// TIA Portal V15.1 export
// export: Created 2024-06-21T08:41:25.533852Z, ExportSetting WithDefaults, DisplayName Totally Integrated Automation Portal, DisplayVersion V15.1 Update 5, DisplayName TIA Portal Openness, DisplayVersion V15.1 Update 5, DisplayName SINAMICS Startdrive Advanced, DisplayVersion V15.1, DisplayName G130, G150, S120, S150, SINAMICS MV, S210, DisplayVersion V15.1, DisplayName G110M, G120, G120C, G120D, G120P, DisplayVersion V15.1, DisplayName STEP 7 Professional, DisplayVersion V15.1 Update 5, DisplayName STEP 7 Safety, DisplayVersion V15.1, DisplayName WinCC Professional, DisplayVersion V15.1 Update 5, DisplayName SIMATIC Visualization Architect, DisplayVersion V15.1
FUNCTION "PNComPLC308" : Void   // FC260, FBD
TITLE = PNComPLC308
{ S7_Optimized_Access := 'FALSE' }
AUTHOR : VCG
FAMILY : LocFncGn
NAME : 211Intf
VERSION : 0.1
// stored: AutoNumber false, IsIECCheckEnabled false, SetENOAutomatically False, UDAEnableTagReadback false
   VAR_OUTPUT
      O_AlarmA : Bool;   // Alarm A
      O_AlarmB : Bool;   // Alarm B
      O_AlarmC : Bool;   // Alarm C
      O_AlarmD : Bool;   // Alarm D
      O_AlarmABCondition : Bool;   // Alarms resetable
      H_IAnim : Word;   // For animation of icon
   END_VAR
BEGIN

REGION Network 1: **** --------------------- 308240CR27 --> 210CR21 --------------------- ****
END_REGION

REGION Network 2: **** 1 - Inputs **** 308230ZS01 - Access Stop Request
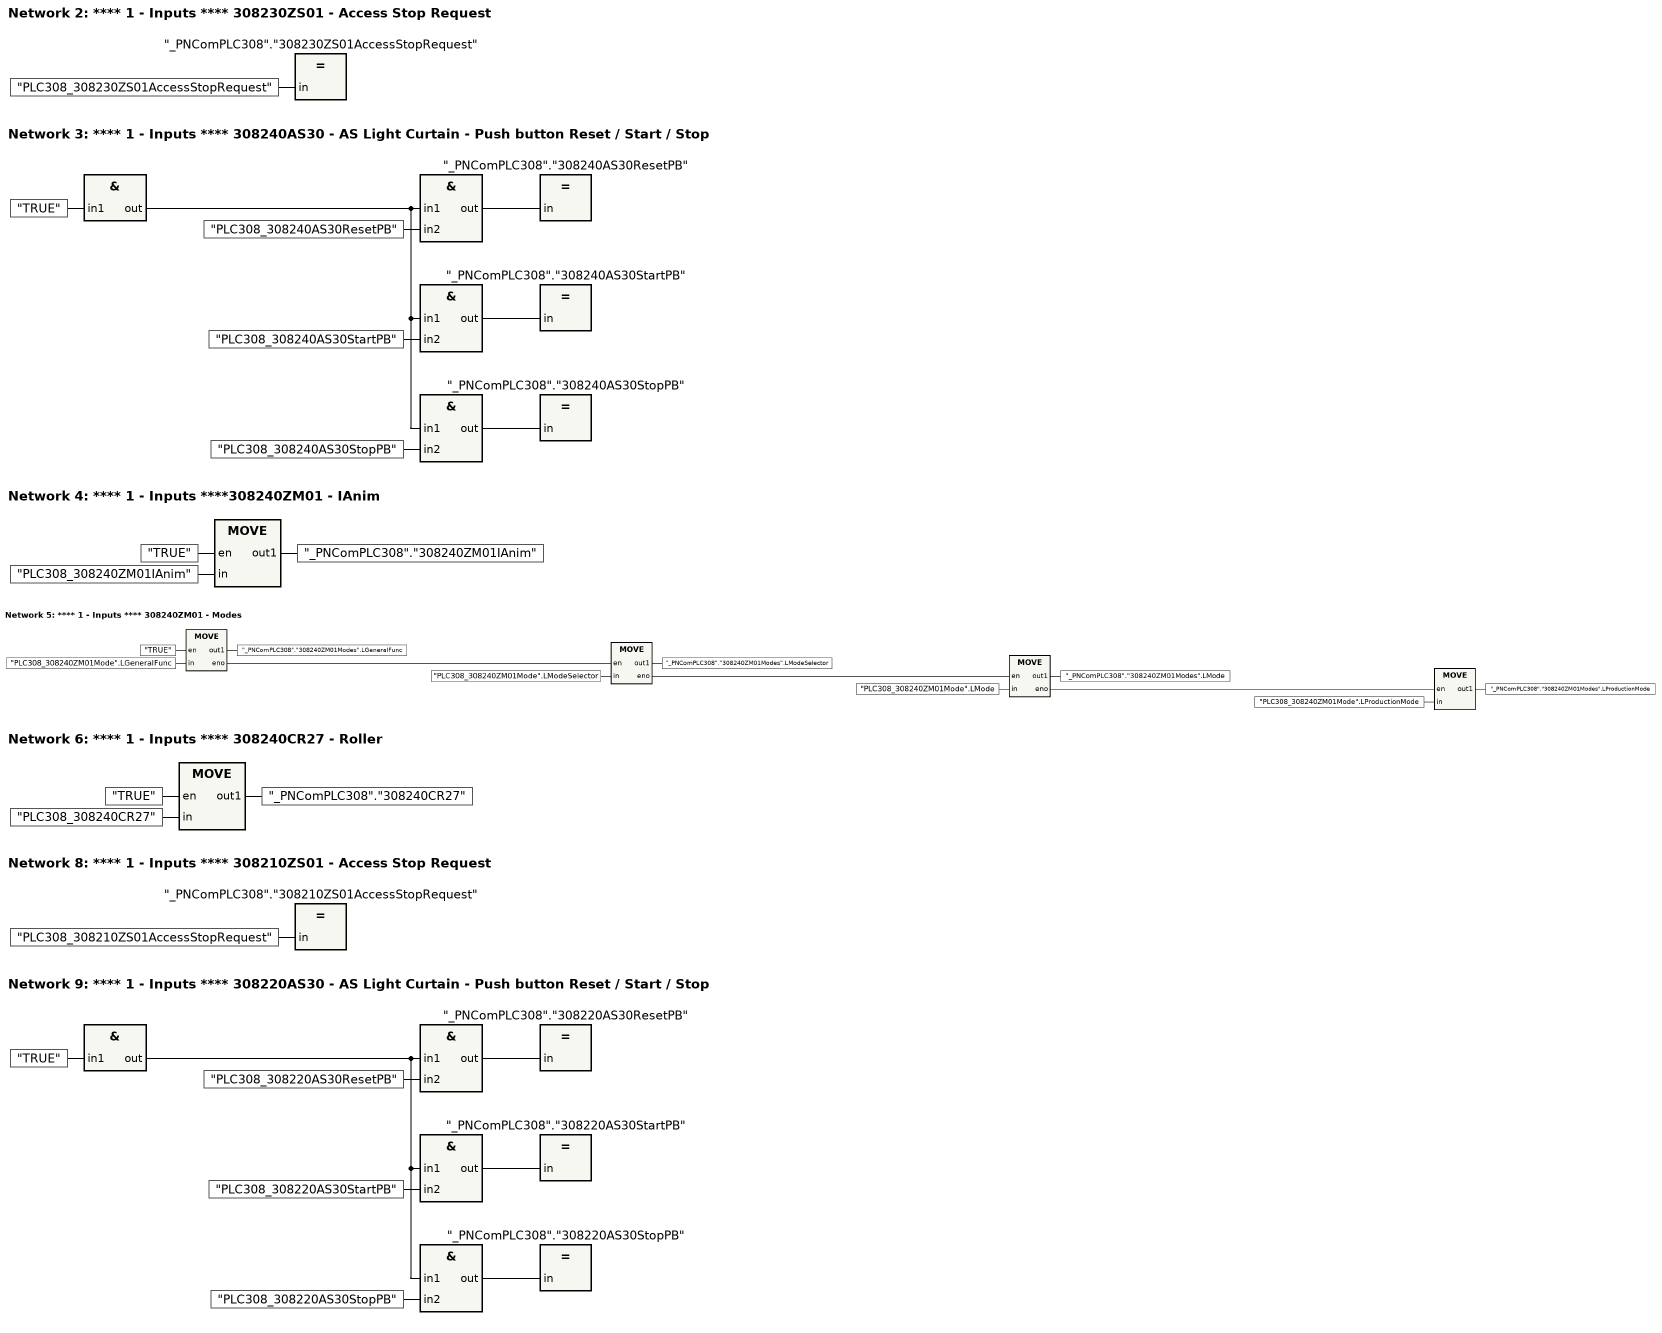
   "_PNComPLC308"."308230ZS01AccessStopRequest" := "PLC308_308230ZS01AccessStopRequest";
END_REGION

REGION Network 3: **** 1 - Inputs **** 308240AS30 - AS Light Curtain - Push button Reset / Start / Stop
   "_PNComPLC308"."308240AS30ResetPB" := "TRUE" AND "PLC308_308240AS30ResetPB";
   "_PNComPLC308"."308240AS30StartPB" := "TRUE" AND "PLC308_308240AS30StartPB";
   "_PNComPLC308"."308240AS30StopPB" := "TRUE" AND "PLC308_308240AS30StopPB";
END_REGION

REGION Network 4: **** 1 - Inputs ****308240ZM01 - IAnim
   IF "TRUE" THEN "_PNComPLC308"."308240ZM01IAnim" := "PLC308_308240ZM01IAnim"; END_IF;
END_REGION

REGION Network 5: **** 1 - Inputs **** 308240ZM01 - Modes
   IF "TRUE" THEN
       "_PNComPLC308"."308240ZM01Modes".LGeneralFunc := "PLC308_308240ZM01Mode".LGeneralFunc;
       "_PNComPLC308"."308240ZM01Modes".LModeSelector := "PLC308_308240ZM01Mode".LModeSelector;
       "_PNComPLC308"."308240ZM01Modes".LMode := "PLC308_308240ZM01Mode".LMode;
       "_PNComPLC308"."308240ZM01Modes".LProductionMode := "PLC308_308240ZM01Mode".LProductionMode;
   END_IF;
END_REGION

REGION Network 6: **** 1 - Inputs **** 308240CR27 - Roller
   IF "TRUE" THEN "_PNComPLC308"."308240CR27" := "PLC308_308240CR27"; END_IF;
END_REGION

REGION Network 7: **** --------------------- 308220CR28 --> 220CR21 --------------------- ****
END_REGION

REGION Network 8: **** 1 - Inputs **** 308210ZS01 - Access Stop Request
   "_PNComPLC308"."308210ZS01AccessStopRequest" := "PLC308_308210ZS01AccessStopRequest";
END_REGION

REGION Network 9: **** 1 - Inputs **** 308220AS30 - AS Light Curtain - Push button Reset / Start / Stop
   "_PNComPLC308"."308220AS30ResetPB" := "TRUE" AND "PLC308_308220AS30ResetPB";
   "_PNComPLC308"."308220AS30StartPB" := "TRUE" AND "PLC308_308220AS30StartPB";
   "_PNComPLC308"."308220AS30StopPB" := "TRUE" AND "PLC308_308220AS30StopPB";
END_REGION

REGION Network 10: **** 1 - Inputs ****308220ZM01 - IAnim
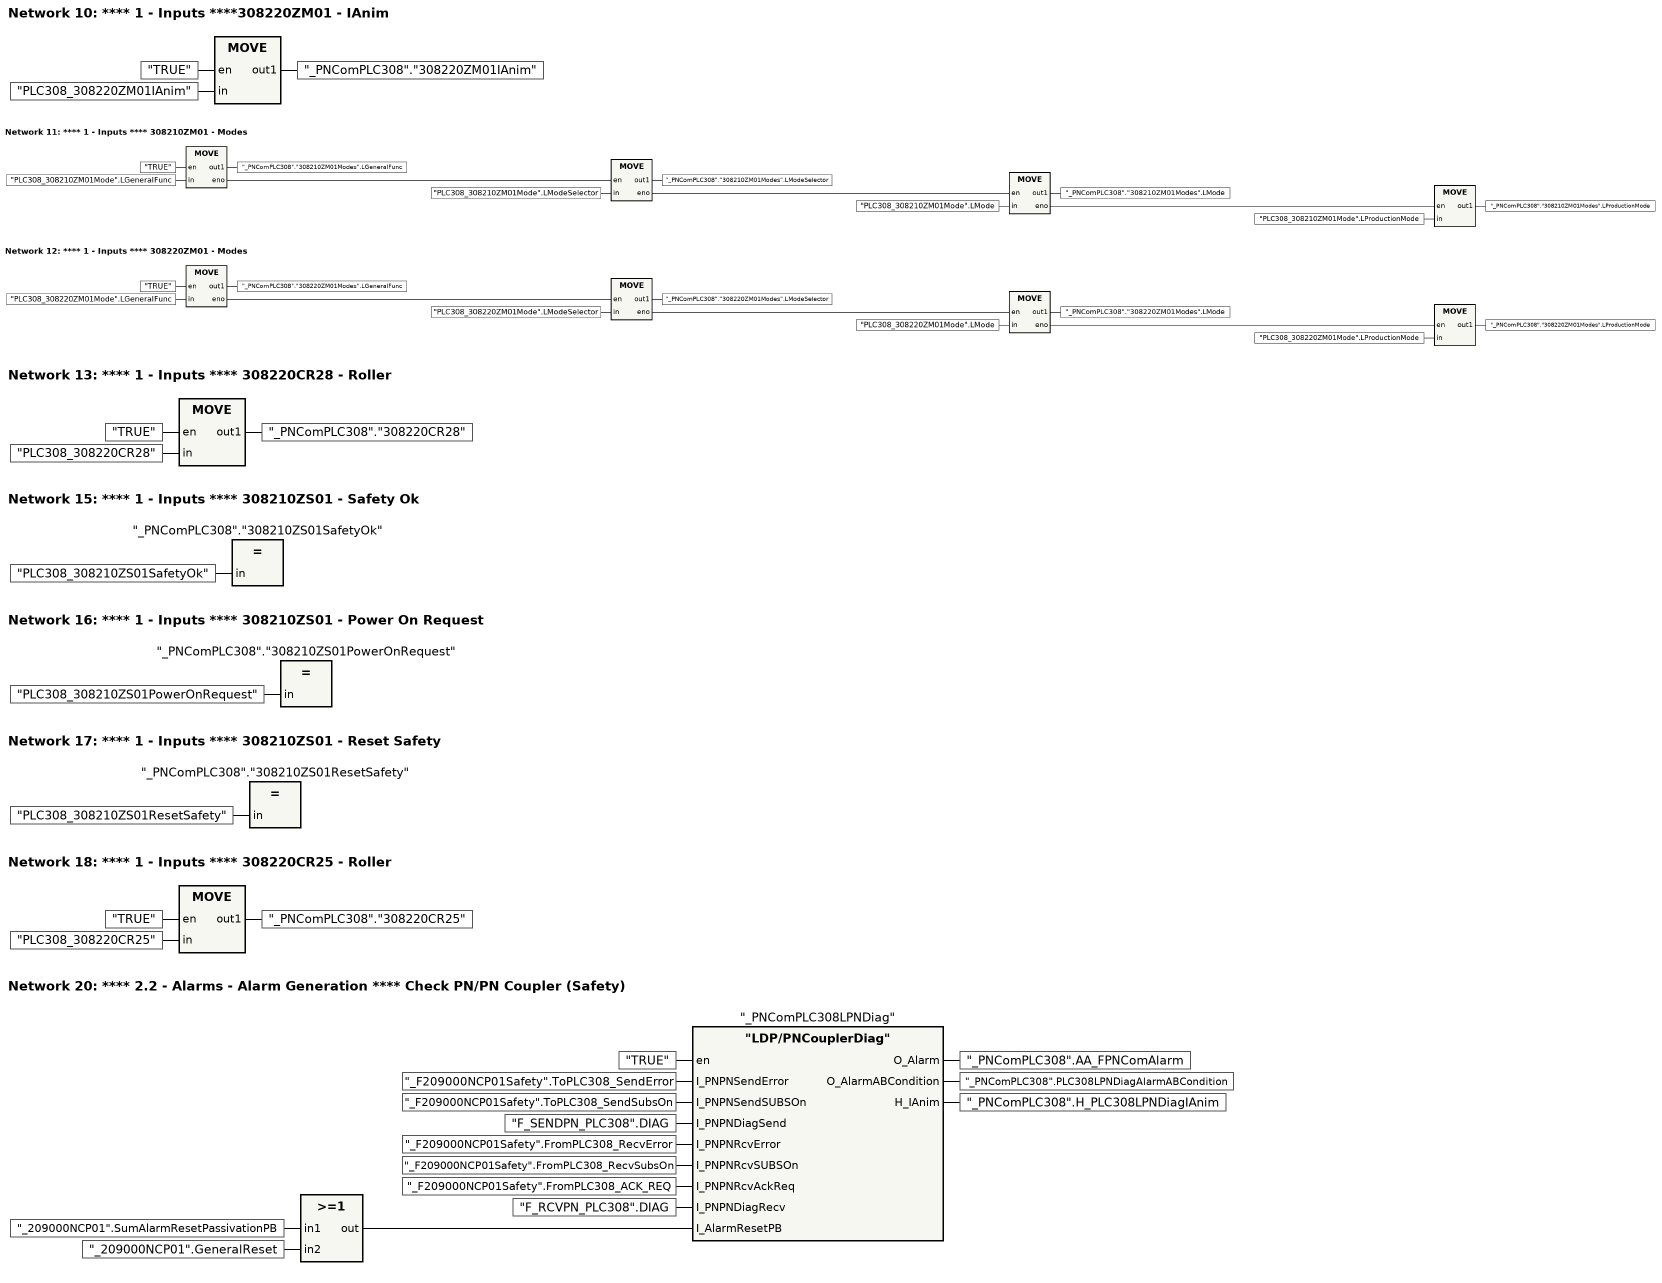
   IF "TRUE" THEN "_PNComPLC308"."308220ZM01IAnim" := "PLC308_308220ZM01IAnim"; END_IF;
END_REGION

REGION Network 11: **** 1 - Inputs **** 308210ZM01 - Modes
   IF "TRUE" THEN
       "_PNComPLC308"."308210ZM01Modes".LGeneralFunc := "PLC308_308210ZM01Mode".LGeneralFunc;
       "_PNComPLC308"."308210ZM01Modes".LModeSelector := "PLC308_308210ZM01Mode".LModeSelector;
       "_PNComPLC308"."308210ZM01Modes".LMode := "PLC308_308210ZM01Mode".LMode;
       "_PNComPLC308"."308210ZM01Modes".LProductionMode := "PLC308_308210ZM01Mode".LProductionMode;
   END_IF;
END_REGION

REGION Network 12: **** 1 - Inputs **** 308220ZM01 - Modes
   IF "TRUE" THEN
       "_PNComPLC308"."308220ZM01Modes".LGeneralFunc := "PLC308_308220ZM01Mode".LGeneralFunc;
       "_PNComPLC308"."308220ZM01Modes".LModeSelector := "PLC308_308220ZM01Mode".LModeSelector;
       "_PNComPLC308"."308220ZM01Modes".LMode := "PLC308_308220ZM01Mode".LMode;
       "_PNComPLC308"."308220ZM01Modes".LProductionMode := "PLC308_308220ZM01Mode".LProductionMode;
   END_IF;
END_REGION

REGION Network 13: **** 1 - Inputs **** 308220CR28 - Roller
   IF "TRUE" THEN "_PNComPLC308"."308220CR28" := "PLC308_308220CR28"; END_IF;
END_REGION

REGION Network 14: **** --------------------- 308220CR25 --> 230CR22 --------------------- ****
END_REGION

REGION Network 15: **** 1 - Inputs **** 308210ZS01 - Safety Ok
   "_PNComPLC308"."308210ZS01SafetyOk" := "PLC308_308210ZS01SafetyOk";
END_REGION

REGION Network 16: **** 1 - Inputs **** 308210ZS01 - Power On Request
   "_PNComPLC308"."308210ZS01PowerOnRequest" := "PLC308_308210ZS01PowerOnRequest";
END_REGION

REGION Network 17: **** 1 - Inputs **** 308210ZS01 - Reset Safety
   "_PNComPLC308"."308210ZS01ResetSafety" := "PLC308_308210ZS01ResetSafety";
END_REGION

REGION Network 18: **** 1 - Inputs **** 308220CR25 - Roller
   IF "TRUE" THEN "_PNComPLC308"."308220CR25" := "PLC308_308220CR25"; END_IF;
END_REGION

REGION Network 19: **** -------------------------------------------------- ****
END_REGION

REGION Network 20: **** 2.2 - Alarms - Alarm Generation **** Check PN/PN Coupler (Safety)
   // Check PN/PN Coupler (Safety)
   IF "TRUE" THEN
       "_PNComPLC308LPNDiag"(I_PNPNSendError := "_F209000NCP01Safety".ToPLC308_SendError,   // "LDP/PNCouplerDiag"
                             I_PNPNSendSUBSOn := "_F209000NCP01Safety".ToPLC308_SendSubsOn,
                             I_PNPNDiagSend := "F_SENDPN_PLC308".DIAG,
                             I_PNPNRcvError := "_F209000NCP01Safety".FromPLC308_RecvError,
                             I_PNPNRcvSUBSOn := "_F209000NCP01Safety".FromPLC308_RecvSubsOn,
                             I_PNPNRcvAckReq := "_F209000NCP01Safety".FromPLC308_ACK_REQ,
                             I_PNPNDiagRecv := "F_RCVPN_PLC308".DIAG,
                             I_AlarmResetPB := "_209000NCP01".SumAlarmResetPassivationPB OR "_209000NCP01".GeneralReset,
                             O_Alarm => "_PNComPLC308".AA_FPNComAlarm,
                             O_AlarmABCondition => "_PNComPLC308".PLC308LPNDiagAlarmABCondition,
                             H_IAnim => "_PNComPLC308".H_PLC308LPNDiagIAnim);
   END_IF;
END_REGION

REGION Network 21: **** 4.6 Machine status - Indication **** Animation In Bit 0_15
   // H_In0_15Anim
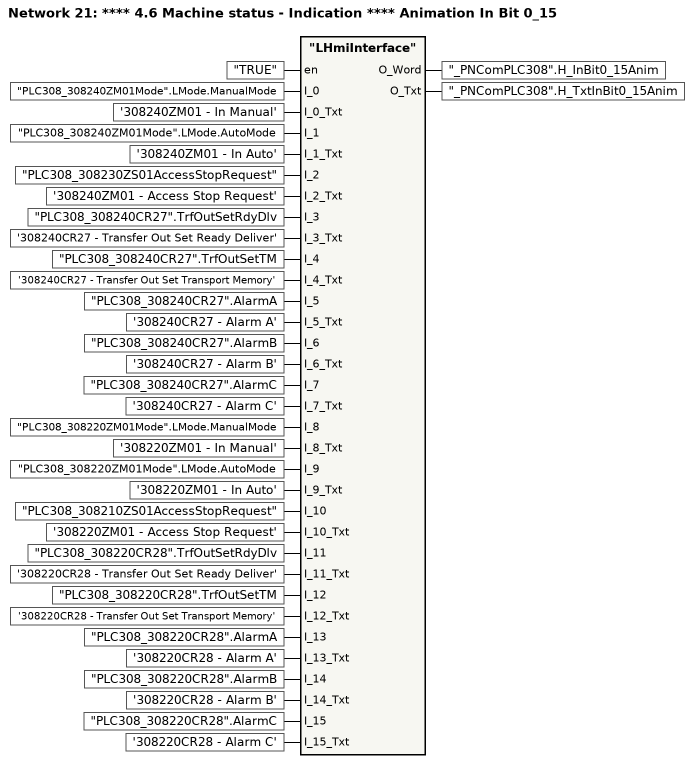
   IF "TRUE" THEN
       "LHmiInterface"(I_0 := "PLC308_308240ZM01Mode".LMode.ManualMode,
                       I_0_Txt := '308240ZM01 - In Manual',
                       I_1 := "PLC308_308240ZM01Mode".LMode.AutoMode,
                       I_1_Txt := '308240ZM01 - In Auto',
                       I_2 := "PLC308_308230ZS01AccessStopRequest",
                       I_2_Txt := '308240ZM01 - Access Stop Request',
                       I_3 := "PLC308_308240CR27".TrfOutSetRdyDlv,
                       I_3_Txt := '308240CR27 - Transfer Out Set Ready Deliver',
                       I_4 := "PLC308_308240CR27".TrfOutSetTM,
                       I_4_Txt := '308240CR27 - Transfer Out Set Transport Memory',
                       I_5 := "PLC308_308240CR27".AlarmA,
                       I_5_Txt := '308240CR27 - Alarm A',
                       I_6 := "PLC308_308240CR27".AlarmB,
                       I_6_Txt := '308240CR27 - Alarm B',
                       I_7 := "PLC308_308240CR27".AlarmC,
                       I_7_Txt := '308240CR27 - Alarm C',
                       I_8 := "PLC308_308220ZM01Mode".LMode.ManualMode,
                       I_8_Txt := '308220ZM01 - In Manual',
                       I_9 := "PLC308_308220ZM01Mode".LMode.AutoMode,
                       I_9_Txt := '308220ZM01 - In Auto',
                       I_10 := "PLC308_308210ZS01AccessStopRequest",
                       I_10_Txt := '308220ZM01 - Access Stop Request',
                       I_11 := "PLC308_308220CR28".TrfOutSetRdyDlv,
                       I_11_Txt := '308220CR28 - Transfer Out Set Ready Deliver',
                       I_12 := "PLC308_308220CR28".TrfOutSetTM,
                       I_12_Txt := '308220CR28 - Transfer Out Set Transport Memory',
                       I_13 := "PLC308_308220CR28".AlarmA,
                       I_13_Txt := '308220CR28 - Alarm A',
                       I_14 := "PLC308_308220CR28".AlarmB,
                       I_14_Txt := '308220CR28 - Alarm B',
                       I_15 := "PLC308_308220CR28".AlarmC,
                       I_15_Txt := '308220CR28 - Alarm C',
                       O_Word => "_PNComPLC308".H_InBit0_15Anim,
                       O_Txt => "_PNComPLC308".H_TxtInBit0_15Anim);
   END_IF;
END_REGION

REGION Network 22: **** 4.6 Machine status - Indication **** Animation In Bit 16_31
   // H_In16_31Anim
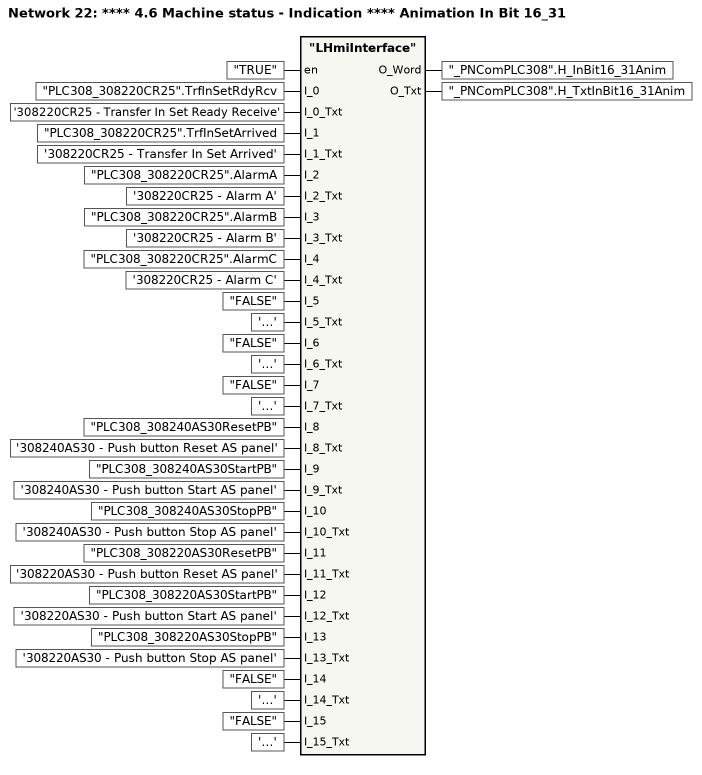
   IF "TRUE" THEN
       "LHmiInterface"(I_0 := "PLC308_308220CR25".TrfInSetRdyRcv,
                       I_0_Txt := '308220CR25 - Transfer In Set Ready Receive',
                       I_1 := "PLC308_308220CR25".TrfInSetArrived,
                       I_1_Txt := '308220CR25 - Transfer In Set Arrived',
                       I_2 := "PLC308_308220CR25".AlarmA,
                       I_2_Txt := '308220CR25 - Alarm A',
                       I_3 := "PLC308_308220CR25".AlarmB,
                       I_3_Txt := '308220CR25 - Alarm B',
                       I_4 := "PLC308_308220CR25".AlarmC,
                       I_4_Txt := '308220CR25 - Alarm C',
                       I_5 := "FALSE",
                       I_5_Txt := '...',
                       I_6 := "FALSE",
                       I_6_Txt := '...',
                       I_7 := "FALSE",
                       I_7_Txt := '...',
                       I_8 := "PLC308_308240AS30ResetPB",
                       I_8_Txt := '308240AS30 - Push button Reset AS panel',
                       I_9 := "PLC308_308240AS30StartPB",
                       I_9_Txt := '308240AS30 - Push button Start AS panel',
                       I_10 := "PLC308_308240AS30StopPB",
                       I_10_Txt := '308240AS30 - Push button Stop AS panel',
                       I_11 := "PLC308_308220AS30ResetPB",
                       I_11_Txt := '308220AS30 - Push button Reset AS panel',
                       I_12 := "PLC308_308220AS30StartPB",
                       I_12_Txt := '308220AS30 - Push button Start AS panel',
                       I_13 := "PLC308_308220AS30StopPB",
                       I_13_Txt := '308220AS30 - Push button Stop AS panel',
                       I_14 := "FALSE",
                       I_14_Txt := '...',
                       I_15 := "FALSE",
                       I_15_Txt := '...',
                       O_Word => "_PNComPLC308".H_InBit16_31Anim,
                       O_Txt => "_PNComPLC308".H_TxtInBit16_31Anim);
   END_IF;
END_REGION

REGION Network 23: **** 4.6 Machine status - Indication **** Animation Out Bit 0_15
   // H_Out0_15Anim
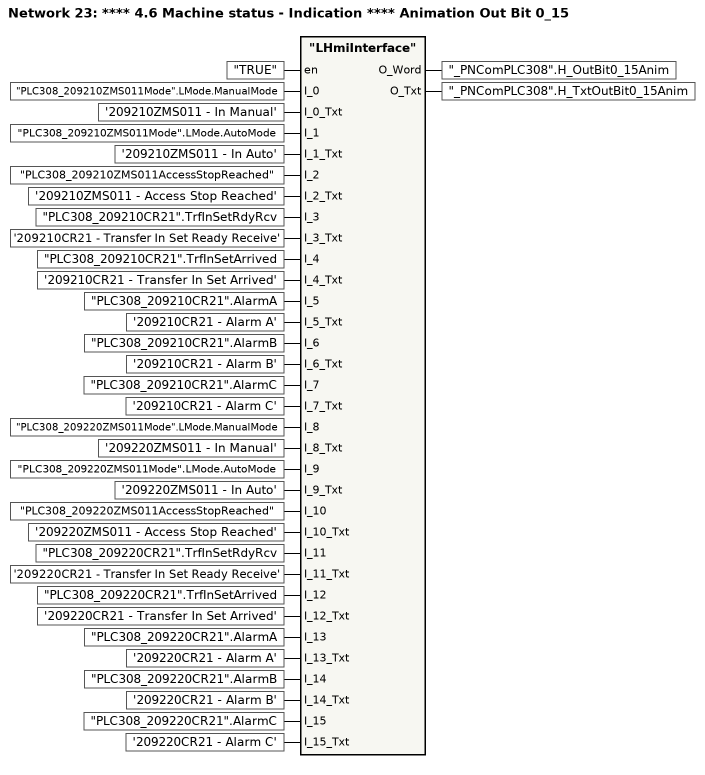
   IF "TRUE" THEN
       "LHmiInterface"(I_0 := "PLC308_209210ZMS011Mode".LMode.ManualMode,
                       I_0_Txt := '209210ZMS011 - In Manual',
                       I_1 := "PLC308_209210ZMS011Mode".LMode.AutoMode,
                       I_1_Txt := '209210ZMS011 - In Auto',
                       I_2 := "PLC308_209210ZMS011AccessStopReached",
                       I_2_Txt := '209210ZMS011 - Access Stop Reached',
                       I_3 := "PLC308_209210CR21".TrfInSetRdyRcv,
                       I_3_Txt := '209210CR21 - Transfer In Set Ready Receive',
                       I_4 := "PLC308_209210CR21".TrfInSetArrived,
                       I_4_Txt := '209210CR21 - Transfer In Set Arrived',
                       I_5 := "PLC308_209210CR21".AlarmA,
                       I_5_Txt := '209210CR21 - Alarm A',
                       I_6 := "PLC308_209210CR21".AlarmB,
                       I_6_Txt := '209210CR21 - Alarm B',
                       I_7 := "PLC308_209210CR21".AlarmC,
                       I_7_Txt := '209210CR21 - Alarm C',
                       I_8 := "PLC308_209220ZMS011Mode".LMode.ManualMode,
                       I_8_Txt := '209220ZMS011 - In Manual',
                       I_9 := "PLC308_209220ZMS011Mode".LMode.AutoMode,
                       I_9_Txt := '209220ZMS011 - In Auto',
                       I_10 := "PLC308_209220ZMS011AccessStopReached",
                       I_10_Txt := '209220ZMS011 - Access Stop Reached',
                       I_11 := "PLC308_209220CR21".TrfInSetRdyRcv,
                       I_11_Txt := '209220CR21 - Transfer In Set Ready Receive',
                       I_12 := "PLC308_209220CR21".TrfInSetArrived,
                       I_12_Txt := '209220CR21 - Transfer In Set Arrived',
                       I_13 := "PLC308_209220CR21".AlarmA,
                       I_13_Txt := '209220CR21 - Alarm A',
                       I_14 := "PLC308_209220CR21".AlarmB,
                       I_14_Txt := '209220CR21 - Alarm B',
                       I_15 := "PLC308_209220CR21".AlarmC,
                       I_15_Txt := '209220CR21 - Alarm C',
                       O_Word => "_PNComPLC308".H_OutBit0_15Anim,
                       O_Txt => "_PNComPLC308".H_TxtOutBit0_15Anim);
   END_IF;
END_REGION

REGION Network 24: **** 4.6 Machine status - Indication **** Animation Out Bit 16_31
   // H_Out16_31Anim
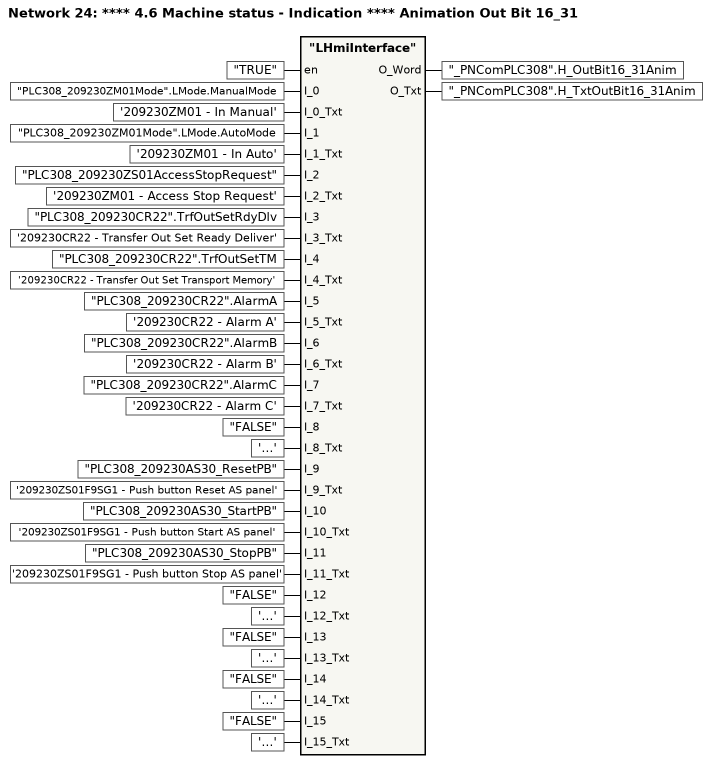
   IF "TRUE" THEN
       "LHmiInterface"(I_0 := "PLC308_209230ZM01Mode".LMode.ManualMode,
                       I_0_Txt := '209230ZM01 - In Manual',
                       I_1 := "PLC308_209230ZM01Mode".LMode.AutoMode,
                       I_1_Txt := '209230ZM01 - In Auto',
                       I_2 := "PLC308_209230ZS01AccessStopRequest",
                       I_2_Txt := '209230ZM01 - Access Stop Request',
                       I_3 := "PLC308_209230CR22".TrfOutSetRdyDlv,
                       I_3_Txt := '209230CR22 - Transfer Out Set Ready Deliver',
                       I_4 := "PLC308_209230CR22".TrfOutSetTM,
                       I_4_Txt := '209230CR22 - Transfer Out Set Transport Memory',
                       I_5 := "PLC308_209230CR22".AlarmA,
                       I_5_Txt := '209230CR22 - Alarm A',
                       I_6 := "PLC308_209230CR22".AlarmB,
                       I_6_Txt := '209230CR22 - Alarm B',
                       I_7 := "PLC308_209230CR22".AlarmC,
                       I_7_Txt := '209230CR22 - Alarm C',
                       I_8 := "FALSE",
                       I_8_Txt := '...',
                       I_9 := "PLC308_209230AS30_ResetPB",
                       I_9_Txt := '209230ZS01F9SG1 - Push button Reset AS panel',
                       I_10 := "PLC308_209230AS30_StartPB",
                       I_10_Txt := '209230ZS01F9SG1 - Push button Start AS panel',
                       I_11 := "PLC308_209230AS30_StopPB",
                       I_11_Txt := '209230ZS01F9SG1 - Push button Stop AS panel',
                       I_12 := "FALSE",
                       I_12_Txt := '...',
                       I_13 := "FALSE",
                       I_13_Txt := '...',
                       I_14 := "FALSE",
                       I_14_Txt := '...',
                       I_15 := "FALSE",
                       I_15_Txt := '...',
                       O_Word => "_PNComPLC308".H_OutBit16_31Anim,
                       O_Txt => "_PNComPLC308".H_TxtOutBit16_31Anim);
   END_IF;
END_REGION

REGION Network 25: **** 4.6 Machine status - Indication **** Animation Safety In Bit 0_15
   // H_FIn0_15Anim
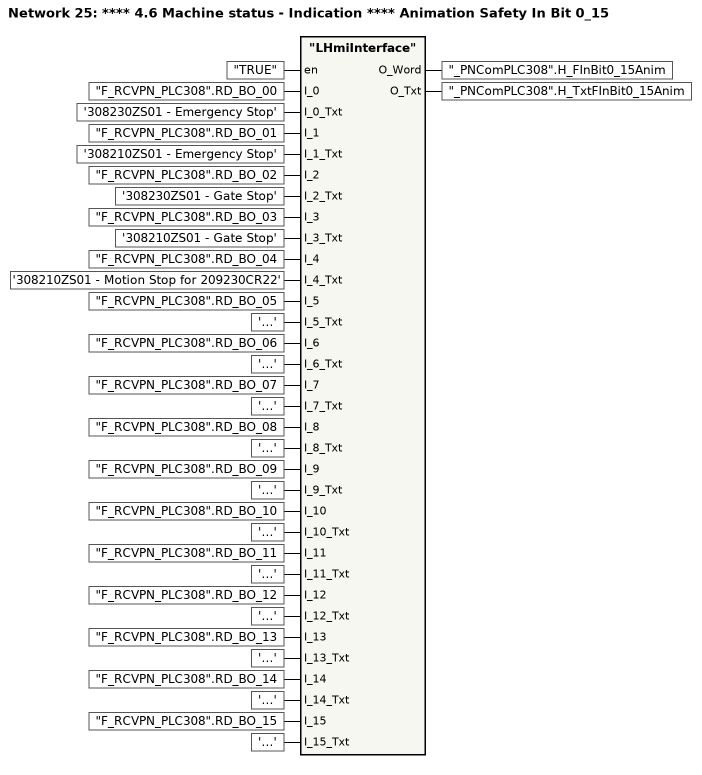
   IF "TRUE" THEN
       "LHmiInterface"(I_0 := "F_RCVPN_PLC308".RD_BO_00,
                       I_0_Txt := '308230ZS01 - Emergency Stop',
                       I_1 := "F_RCVPN_PLC308".RD_BO_01,
                       I_1_Txt := '308210ZS01 - Emergency Stop',
                       I_2 := "F_RCVPN_PLC308".RD_BO_02,
                       I_2_Txt := '308230ZS01 - Gate Stop',
                       I_3 := "F_RCVPN_PLC308".RD_BO_03,
                       I_3_Txt := '308210ZS01 - Gate Stop',
                       I_4 := "F_RCVPN_PLC308".RD_BO_04,
                       I_4_Txt := '308210ZS01 - Motion Stop for 209230CR22',
                       I_5 := "F_RCVPN_PLC308".RD_BO_05,
                       I_5_Txt := '...',
                       I_6 := "F_RCVPN_PLC308".RD_BO_06,
                       I_6_Txt := '...',
                       I_7 := "F_RCVPN_PLC308".RD_BO_07,
                       I_7_Txt := '...',
                       I_8 := "F_RCVPN_PLC308".RD_BO_08,
                       I_8_Txt := '...',
                       I_9 := "F_RCVPN_PLC308".RD_BO_09,
                       I_9_Txt := '...',
                       I_10 := "F_RCVPN_PLC308".RD_BO_10,
                       I_10_Txt := '...',
                       I_11 := "F_RCVPN_PLC308".RD_BO_11,
                       I_11_Txt := '...',
                       I_12 := "F_RCVPN_PLC308".RD_BO_12,
                       I_12_Txt := '...',
                       I_13 := "F_RCVPN_PLC308".RD_BO_13,
                       I_13_Txt := '...',
                       I_14 := "F_RCVPN_PLC308".RD_BO_14,
                       I_14_Txt := '...',
                       I_15 := "F_RCVPN_PLC308".RD_BO_15,
                       I_15_Txt := '...',
                       O_Word => "_PNComPLC308".H_FInBit0_15Anim,
                       O_Txt => "_PNComPLC308".H_TxtFInBit0_15Anim);
   END_IF;
END_REGION

REGION Network 26: **** 4.6 Machine status - Indication **** Animation Safety Out Bit 0_15
   // H_FOut0_15Anim
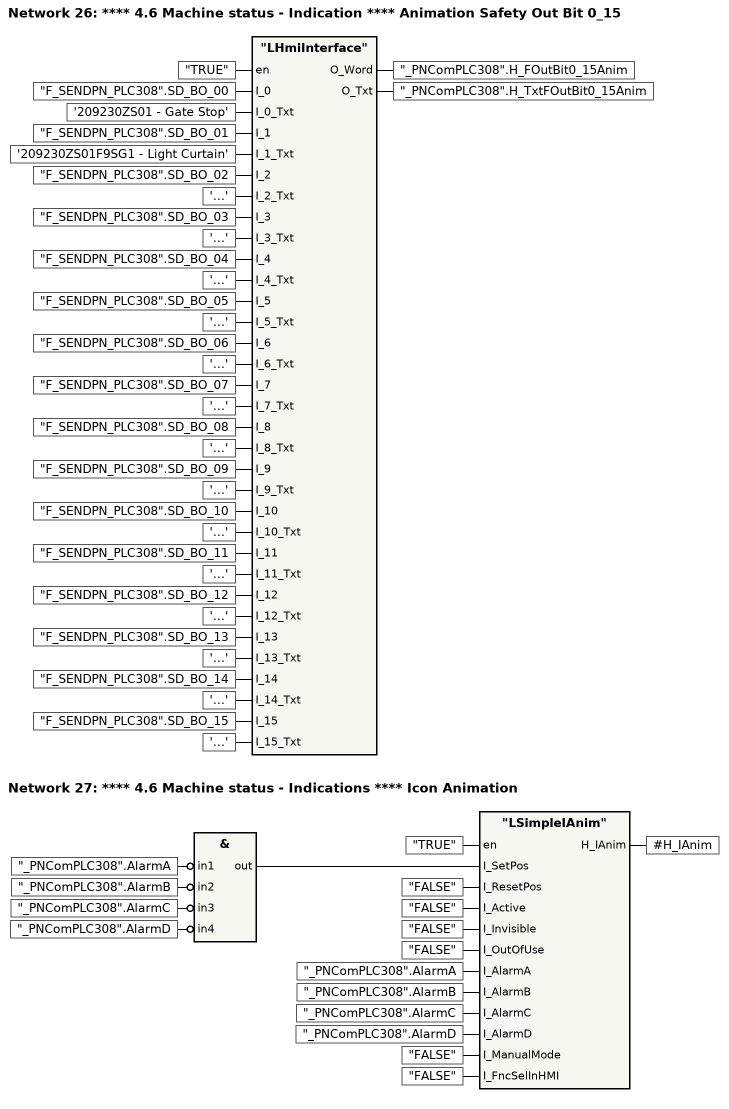
   IF "TRUE" THEN
       "LHmiInterface"(I_0 := "F_SENDPN_PLC308".SD_BO_00,
                       I_0_Txt := '209230ZS01 - Gate Stop',
                       I_1 := "F_SENDPN_PLC308".SD_BO_01,
                       I_1_Txt := '209230ZS01F9SG1 - Light Curtain',
                       I_2 := "F_SENDPN_PLC308".SD_BO_02,
                       I_2_Txt := '...',
                       I_3 := "F_SENDPN_PLC308".SD_BO_03,
                       I_3_Txt := '...',
                       I_4 := "F_SENDPN_PLC308".SD_BO_04,
                       I_4_Txt := '...',
                       I_5 := "F_SENDPN_PLC308".SD_BO_05,
                       I_5_Txt := '...',
                       I_6 := "F_SENDPN_PLC308".SD_BO_06,
                       I_6_Txt := '...',
                       I_7 := "F_SENDPN_PLC308".SD_BO_07,
                       I_7_Txt := '...',
                       I_8 := "F_SENDPN_PLC308".SD_BO_08,
                       I_8_Txt := '...',
                       I_9 := "F_SENDPN_PLC308".SD_BO_09,
                       I_9_Txt := '...',
                       I_10 := "F_SENDPN_PLC308".SD_BO_10,
                       I_10_Txt := '...',
                       I_11 := "F_SENDPN_PLC308".SD_BO_11,
                       I_11_Txt := '...',
                       I_12 := "F_SENDPN_PLC308".SD_BO_12,
                       I_12_Txt := '...',
                       I_13 := "F_SENDPN_PLC308".SD_BO_13,
                       I_13_Txt := '...',
                       I_14 := "F_SENDPN_PLC308".SD_BO_14,
                       I_14_Txt := '...',
                       I_15 := "F_SENDPN_PLC308".SD_BO_15,
                       I_15_Txt := '...',
                       O_Word => "_PNComPLC308".H_FOutBit0_15Anim,
                       O_Txt => "_PNComPLC308".H_TxtFOutBit0_15Anim);
   END_IF;
END_REGION

REGION Network 27: **** 4.6 Machine status - Indications **** Icon Animation
   // Animation for icon
   IF "TRUE" THEN
       "LSimpleIAnim"(I_SetPos := NOT "_PNComPLC308".AlarmA AND NOT "_PNComPLC308".AlarmB AND NOT "_PNComPLC308".AlarmC AND NOT "_PNComPLC308".AlarmD,
                      I_ResetPos := "FALSE",
                      I_Active := "FALSE",
                      I_Invisible := "FALSE",
                      I_OutOfUse := "FALSE",
                      I_AlarmA := "_PNComPLC308".AlarmA,
                      I_AlarmB := "_PNComPLC308".AlarmB,
                      I_AlarmC := "_PNComPLC308".AlarmC,
                      I_AlarmD := "_PNComPLC308".AlarmD,
                      I_ManualMode := "FALSE",
                      I_FncSelInHMI := "FALSE",
                      H_IAnim => #H_IAnim);
   END_IF;
END_REGION

REGION Network 28: **** 4.6 - Machine status - Indications **** Animation
   // Animation
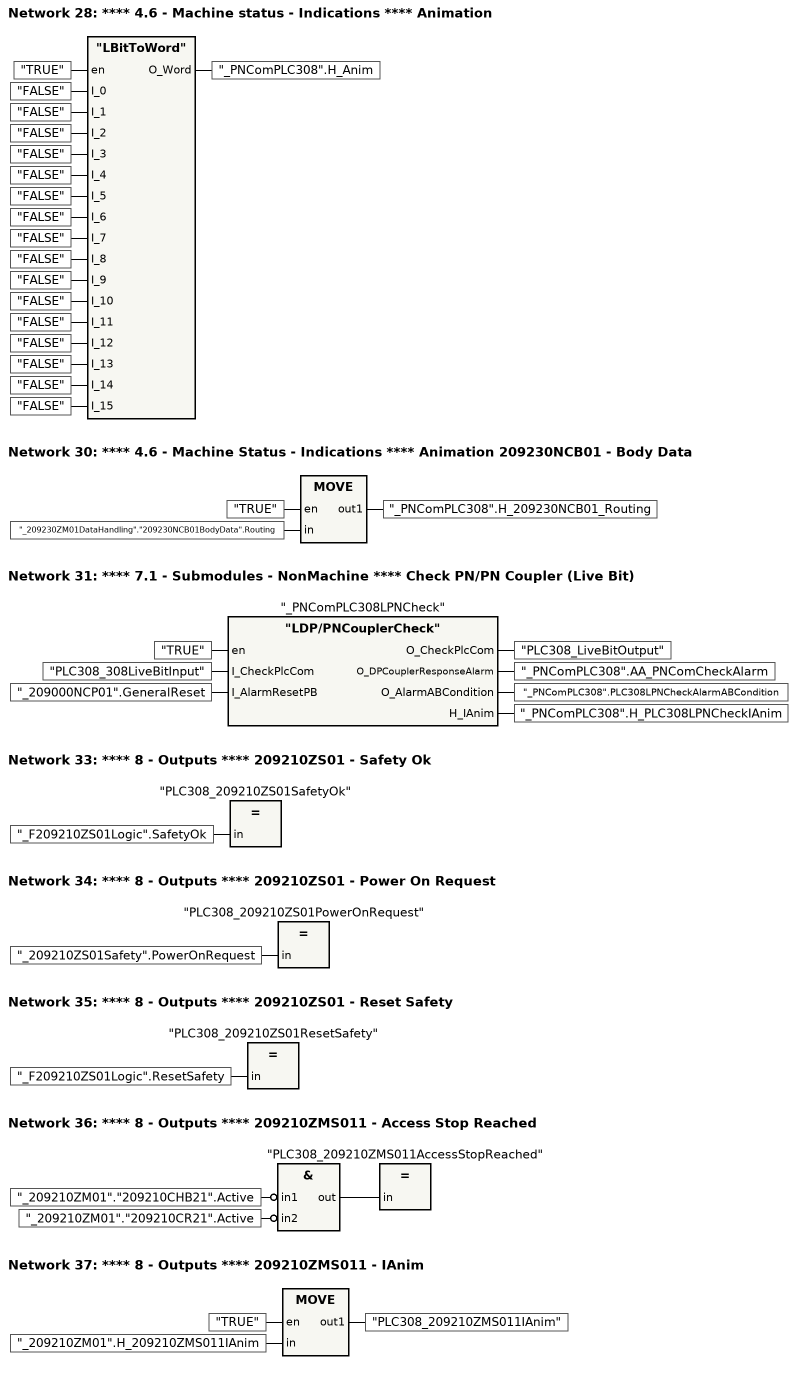
   IF "TRUE" THEN
       "LBitToWord"(I_0 := "FALSE",
                    I_1 := "FALSE",
                    I_2 := "FALSE",
                    I_3 := "FALSE",
                    I_4 := "FALSE",
                    I_5 := "FALSE",
                    I_6 := "FALSE",
                    I_7 := "FALSE",
                    I_8 := "FALSE",
                    I_9 := "FALSE",
                    I_10 := "FALSE",
                    I_11 := "FALSE",
                    I_12 := "FALSE",
                    I_13 := "FALSE",
                    I_14 := "FALSE",
                    I_15 := "FALSE",
                    O_Word => "_PNComPLC308".H_Anim);
   END_IF;
END_REGION

NETWORK
TITLE = **** 4.6 - Machine Status - Indications **** Animation DB number
// DB number
      OPN   "_PNComPLC308";
      L     DBNO;
      T     "_PNComPLC308".H_DBnr;

REGION Network 30: **** 4.6 - Machine Status - Indications **** Animation 209230NCB01 - Body Data
   IF "TRUE" THEN
       "_PNComPLC308".H_209230NCB01_Routing := "_209230ZM01DataHandling"."209230NCB01BodyData".Routing;
   END_IF;
END_REGION

REGION Network 31: **** 7.1 - Submodules - NonMachine **** Check PN/PN Coupler (Live Bit)
   // Check PN/PN Coupler (Live Bit)
   IF "TRUE" THEN
       "_PNComPLC308LPNCheck"(I_CheckPlcCom := "PLC308_308LiveBitInput",   // "LDP/PNCouplerCheck"
                              I_AlarmResetPB := "_209000NCP01".GeneralReset,
                              O_CheckPlcCom => "PLC308_LiveBitOutput",
                              O_DPCouplerResponseAlarm => "_PNComPLC308".AA_PNComCheckAlarm,
                              O_AlarmABCondition => "_PNComPLC308".PLC308LPNCheckAlarmABCondition,
                              H_IAnim => "_PNComPLC308".H_PLC308LPNCheckIAnim);
   END_IF;
END_REGION

REGION Network 32: **** --------------------- 210CR21 --> 308240CR27 --------------------- ****
END_REGION

REGION Network 33: **** 8 - Outputs **** 209210ZS01 - Safety Ok
   "PLC308_209210ZS01SafetyOk" := "_F209210ZS01Logic".SafetyOk;
END_REGION

REGION Network 34: **** 8 - Outputs **** 209210ZS01 - Power On Request
   "PLC308_209210ZS01PowerOnRequest" := "_209210ZS01Safety".PowerOnRequest;
END_REGION

REGION Network 35: **** 8 - Outputs **** 209210ZS01 - Reset Safety
   "PLC308_209210ZS01ResetSafety" := "_F209210ZS01Logic".ResetSafety;
END_REGION

REGION Network 36: **** 8 - Outputs **** 209210ZMS011 - Access Stop Reached
   "PLC308_209210ZMS011AccessStopReached" := NOT "_209210ZM01"."209210CHB21".Active AND NOT "_209210ZM01"."209210CR21".Active;
END_REGION

REGION Network 37: **** 8 - Outputs **** 209210ZMS011 - IAnim
   IF "TRUE" THEN "PLC308_209210ZMS011IAnim" := "_209210ZM01".H_209210ZMS011IAnim; END_IF;
END_REGION

REGION Network 38: **** 8 - Outputs **** 209210ZMS011 - Modes
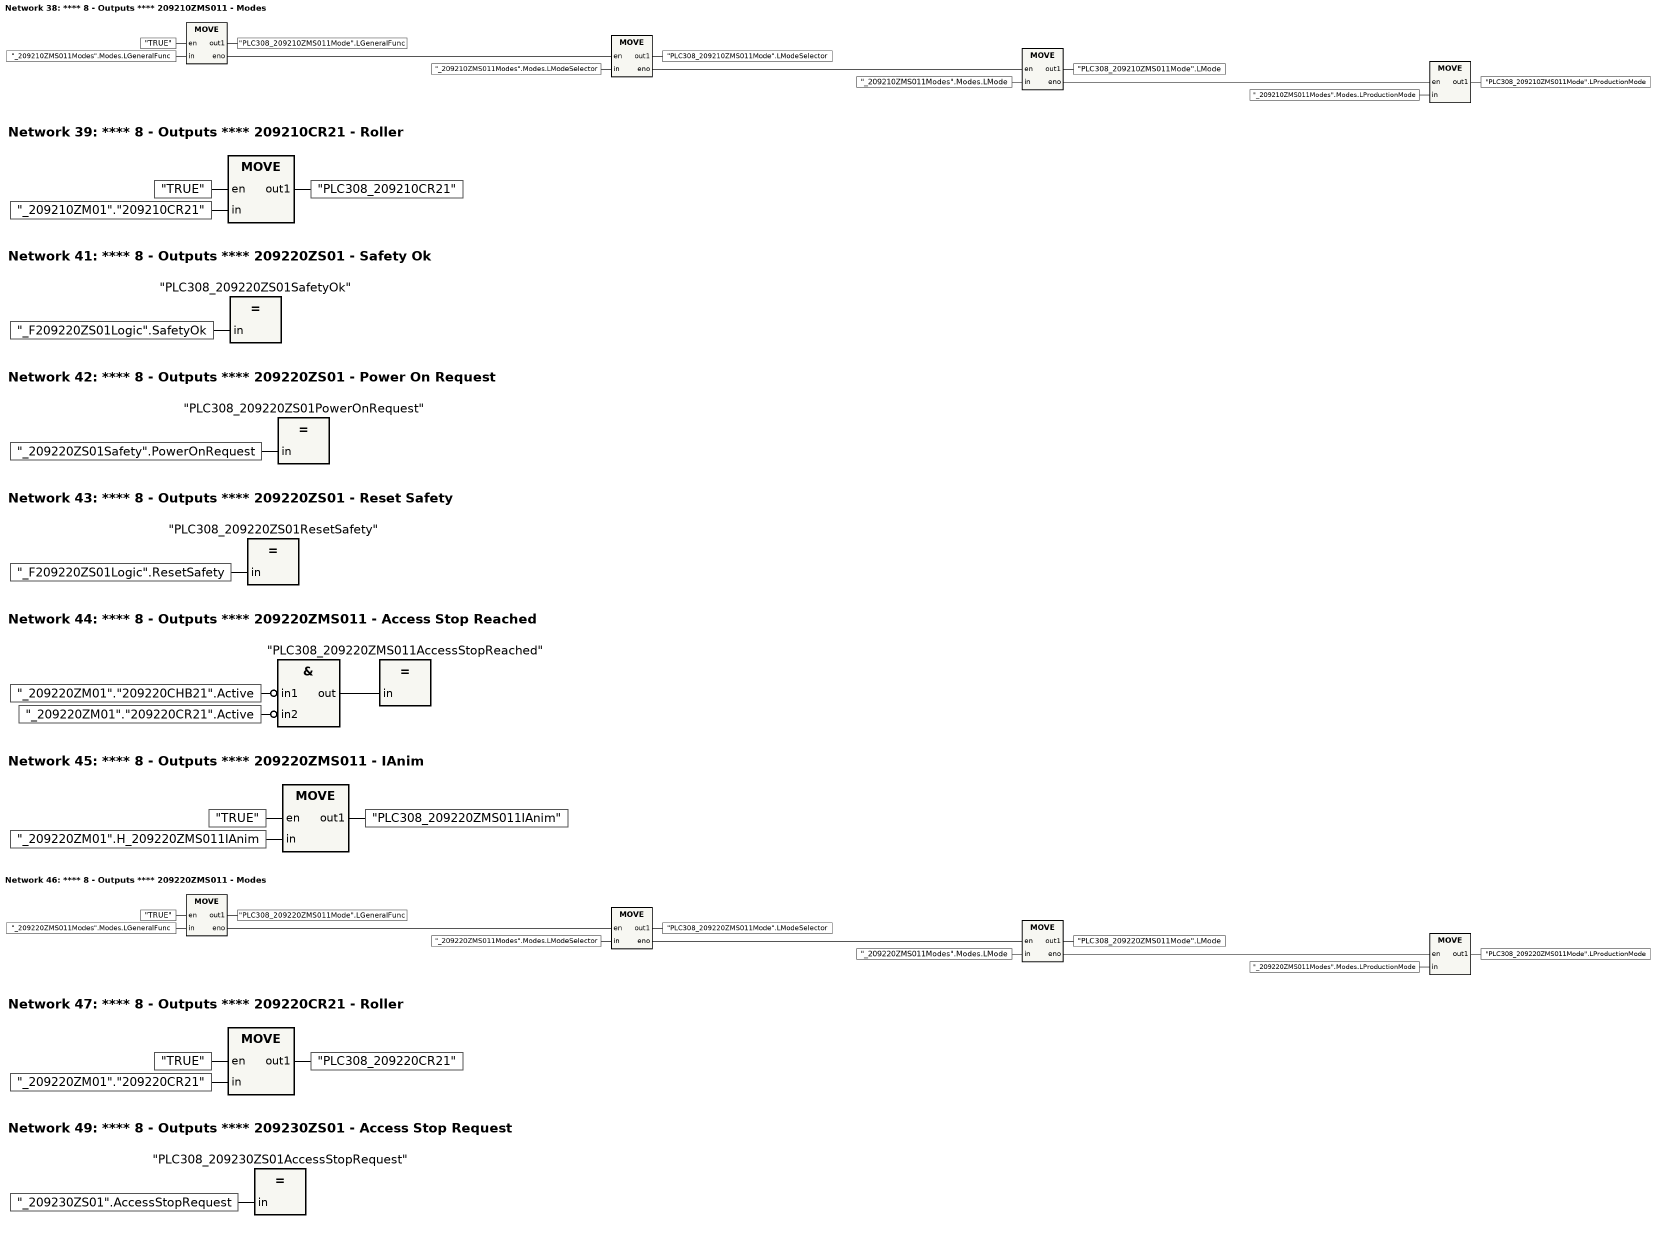
   IF "TRUE" THEN
       "PLC308_209210ZMS011Mode".LGeneralFunc := "_209210ZMS011Modes".Modes.LGeneralFunc;
       "PLC308_209210ZMS011Mode".LModeSelector := "_209210ZMS011Modes".Modes.LModeSelector;
       "PLC308_209210ZMS011Mode".LMode := "_209210ZMS011Modes".Modes.LMode;
       "PLC308_209210ZMS011Mode".LProductionMode := "_209210ZMS011Modes".Modes.LProductionMode;
   END_IF;
END_REGION

REGION Network 39: **** 8 - Outputs **** 209210CR21 - Roller
   IF "TRUE" THEN "PLC308_209210CR21" := "_209210ZM01"."209210CR21"; END_IF;
END_REGION

REGION Network 40: **** --------------------- 220CR21 --> 308220CR28 --------------------- ****
END_REGION

REGION Network 41: **** 8 - Outputs **** 209220ZS01 - Safety Ok
   "PLC308_209220ZS01SafetyOk" := "_F209220ZS01Logic".SafetyOk;
END_REGION

REGION Network 42: **** 8 - Outputs **** 209220ZS01 - Power On Request
   "PLC308_209220ZS01PowerOnRequest" := "_209220ZS01Safety".PowerOnRequest;
END_REGION

REGION Network 43: **** 8 - Outputs **** 209220ZS01 - Reset Safety
   "PLC308_209220ZS01ResetSafety" := "_F209220ZS01Logic".ResetSafety;
END_REGION

REGION Network 44: **** 8 - Outputs **** 209220ZMS011 - Access Stop Reached
   "PLC308_209220ZMS011AccessStopReached" := NOT "_209220ZM01"."209220CHB21".Active AND NOT "_209220ZM01"."209220CR21".Active;
END_REGION

REGION Network 45: **** 8 - Outputs **** 209220ZMS011 - IAnim
   IF "TRUE" THEN "PLC308_209220ZMS011IAnim" := "_209220ZM01".H_209220ZMS011IAnim; END_IF;
END_REGION

REGION Network 46: **** 8 - Outputs **** 209220ZMS011 - Modes
   IF "TRUE" THEN
       "PLC308_209220ZMS011Mode".LGeneralFunc := "_209220ZMS011Modes".Modes.LGeneralFunc;
       "PLC308_209220ZMS011Mode".LModeSelector := "_209220ZMS011Modes".Modes.LModeSelector;
       "PLC308_209220ZMS011Mode".LMode := "_209220ZMS011Modes".Modes.LMode;
       "PLC308_209220ZMS011Mode".LProductionMode := "_209220ZMS011Modes".Modes.LProductionMode;
   END_IF;
END_REGION

REGION Network 47: **** 8 - Outputs **** 209220CR21 - Roller
   IF "TRUE" THEN "PLC308_209220CR21" := "_209220ZM01"."209220CR21"; END_IF;
END_REGION

REGION Network 48: **** --------------------- 230CR22 --> 308220CR25 --------------------- ****
END_REGION

REGION Network 49: **** 8 - Outputs **** 209230ZS01 - Access Stop Request
   "PLC308_209230ZS01AccessStopRequest" := "_209230ZS01".AccessStopRequest;
END_REGION

REGION Network 50: **** 8 - Outputs **** 209230AS30 - AS Light Curtain - Push button Reset / Start / Stop
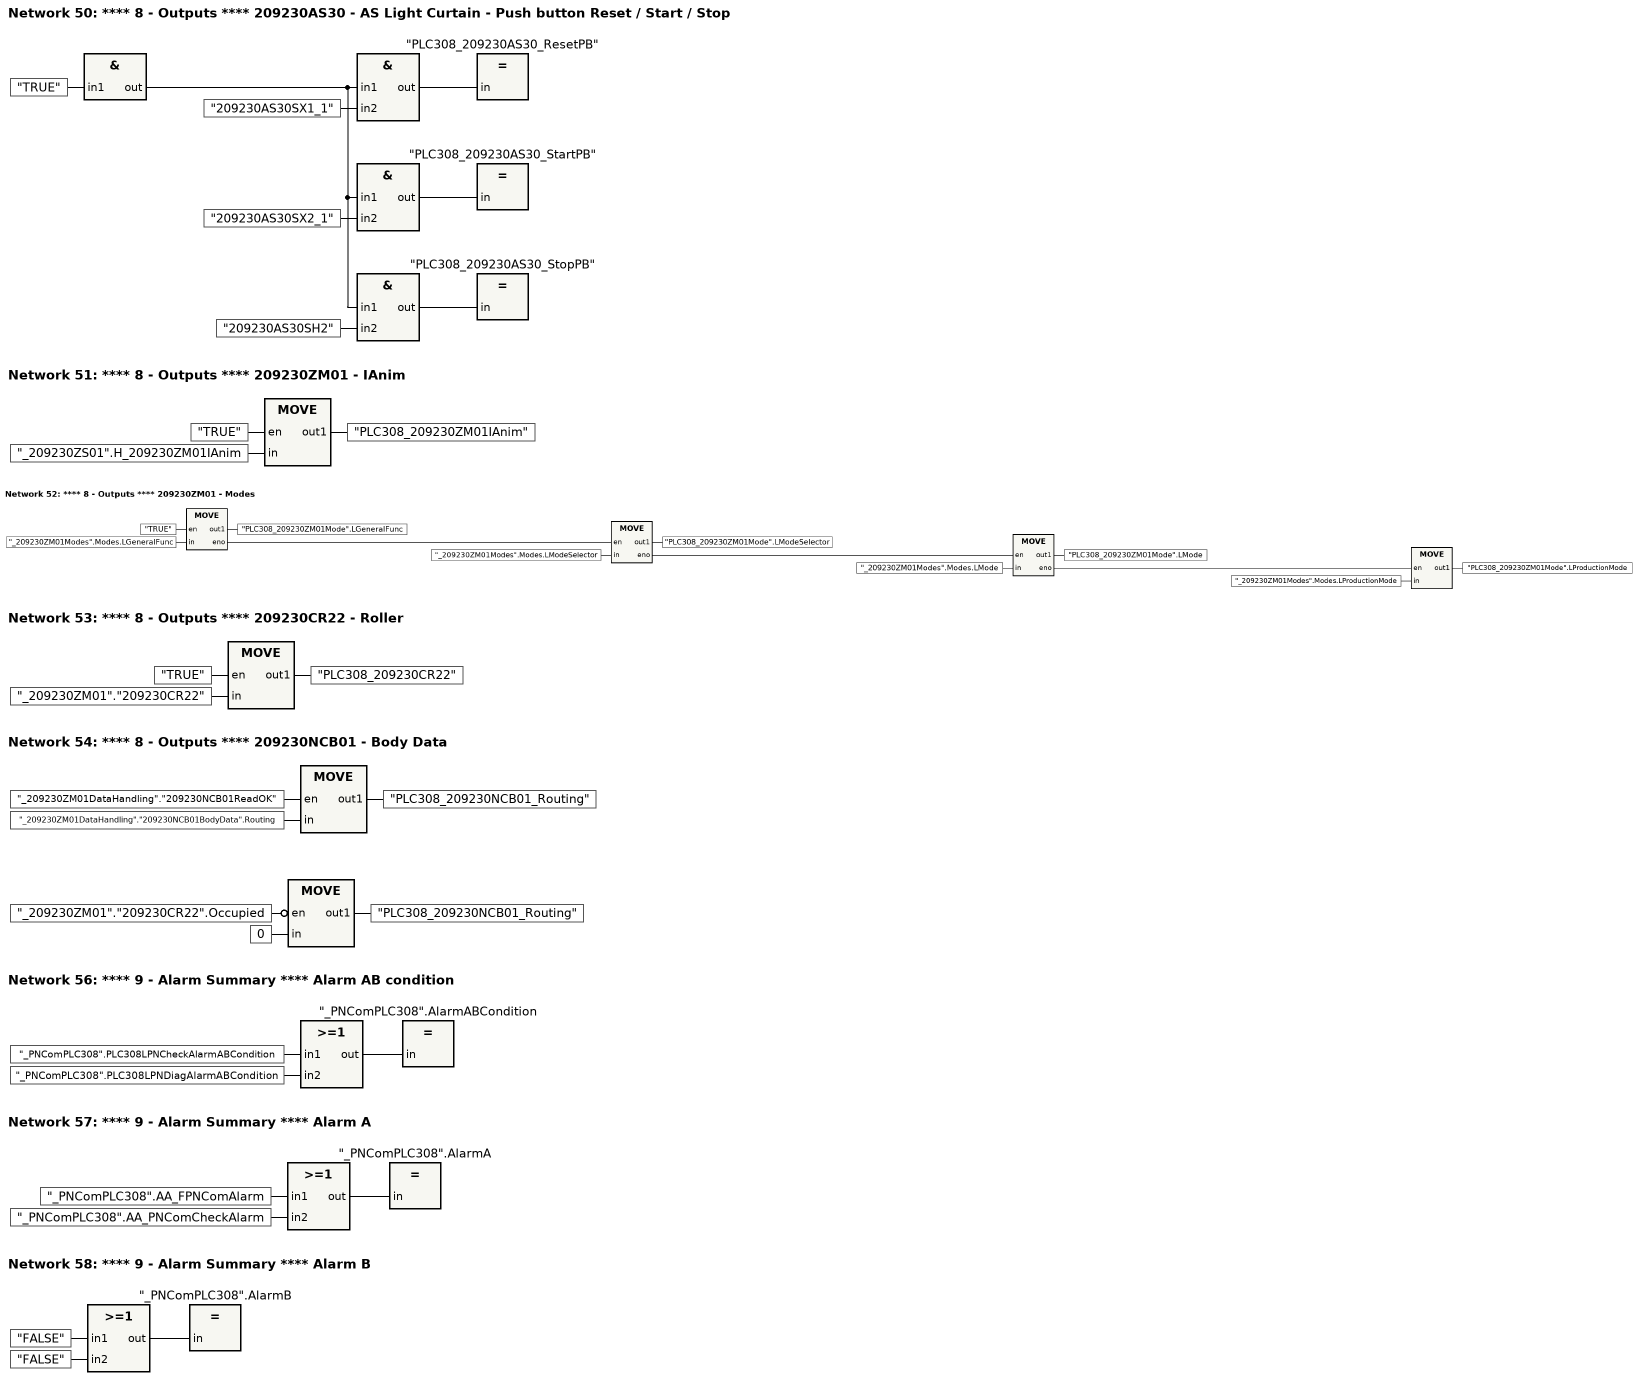
   "PLC308_209230AS30_ResetPB" := "TRUE" AND "209230AS30SX1_1";
   "PLC308_209230AS30_StartPB" := "TRUE" AND "209230AS30SX2_1";
   "PLC308_209230AS30_StopPB" := "TRUE" AND "209230AS30SH2";
END_REGION

REGION Network 51: **** 8 - Outputs **** 209230ZM01 - IAnim
   IF "TRUE" THEN "PLC308_209230ZM01IAnim" := "_209230ZS01".H_209230ZM01IAnim; END_IF;
END_REGION

REGION Network 52: **** 8 - Outputs **** 209230ZM01 - Modes
   IF "TRUE" THEN
       "PLC308_209230ZM01Mode".LGeneralFunc := "_209230ZM01Modes".Modes.LGeneralFunc;
       "PLC308_209230ZM01Mode".LModeSelector := "_209230ZM01Modes".Modes.LModeSelector;
       "PLC308_209230ZM01Mode".LMode := "_209230ZM01Modes".Modes.LMode;
       "PLC308_209230ZM01Mode".LProductionMode := "_209230ZM01Modes".Modes.LProductionMode;
   END_IF;
END_REGION

REGION Network 53: **** 8 - Outputs **** 209230CR22 - Roller
   IF "TRUE" THEN "PLC308_209230CR22" := "_209230ZM01"."209230CR22"; END_IF;
END_REGION

REGION Network 54: **** 8 - Outputs **** 209230NCB01 - Body Data
   IF "_209230ZM01DataHandling"."209230NCB01ReadOK" THEN
       "PLC308_209230NCB01_Routing" := "_209230ZM01DataHandling"."209230NCB01BodyData".Routing;
   END_IF;
   IF NOT "_209230ZM01"."209230CR22".Occupied THEN "PLC308_209230NCB01_Routing" := 0; END_IF;
END_REGION

REGION Network 55: **** -------------------------------------------------- ****
END_REGION

REGION Network 56: **** 9 - Alarm Summary **** Alarm AB condition
   // Alarm AB condition
   "_PNComPLC308".AlarmABCondition := "_PNComPLC308".PLC308LPNCheckAlarmABCondition OR "_PNComPLC308".PLC308LPNDiagAlarmABCondition;
END_REGION

REGION Network 57: **** 9 - Alarm Summary **** Alarm A
   // Summary of alarms A
   "_PNComPLC308".AlarmA := "_PNComPLC308".AA_FPNComAlarm OR "_PNComPLC308".AA_PNComCheckAlarm;
END_REGION

REGION Network 58: **** 9 - Alarm Summary **** Alarm B
   // Summary of alarms B
   "_PNComPLC308".AlarmB := "FALSE" OR "FALSE";
END_REGION

REGION Network 59: **** 9 - Alarm Summary **** Alarm C
   // Summary of alarms C
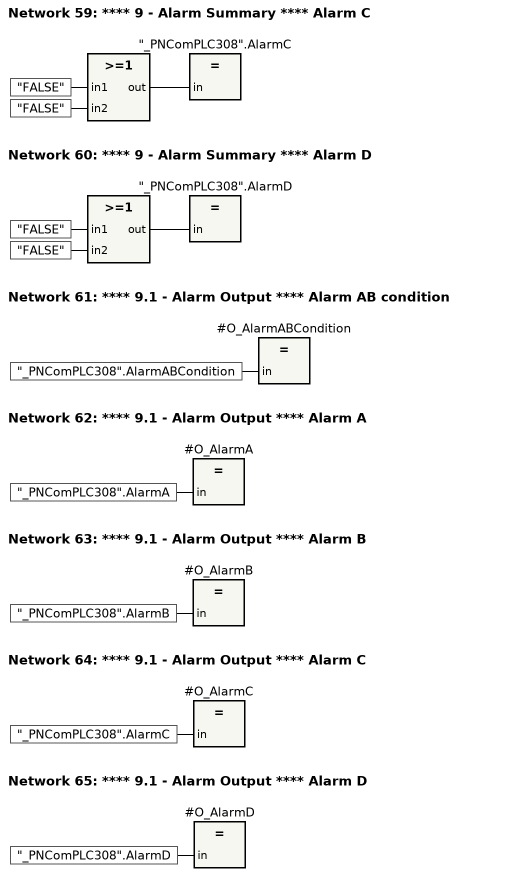
   "_PNComPLC308".AlarmC := "FALSE" OR "FALSE";
END_REGION

REGION Network 60: **** 9 - Alarm Summary **** Alarm D
   // Summary of alarms D
   "_PNComPLC308".AlarmD := "FALSE" OR "FALSE";
END_REGION

REGION Network 61: **** 9.1 - Alarm Output **** Alarm AB condition
   // Alarm AB condition
   #O_AlarmABCondition := "_PNComPLC308".AlarmABCondition;
END_REGION

REGION Network 62: **** 9.1 - Alarm Output **** Alarm A
   // Summary of alarms A
   #O_AlarmA := "_PNComPLC308".AlarmA;
END_REGION

REGION Network 63: **** 9.1 - Alarm Output **** Alarm B
   // Summary of alarms B
   #O_AlarmB := "_PNComPLC308".AlarmB;
END_REGION

REGION Network 64: **** 9.1 - Alarm Output **** Alarm C
   // Summary of alarms C
   #O_AlarmC := "_PNComPLC308".AlarmC;
END_REGION

REGION Network 65: **** 9.1 - Alarm Output **** Alarm D
   // Summary of alarms D
   #O_AlarmD := "_PNComPLC308".AlarmD;
END_REGION

REGION Network 66: **** 9.2 - Alarm DWord**** Alarm To DWord
   // Alarm Word
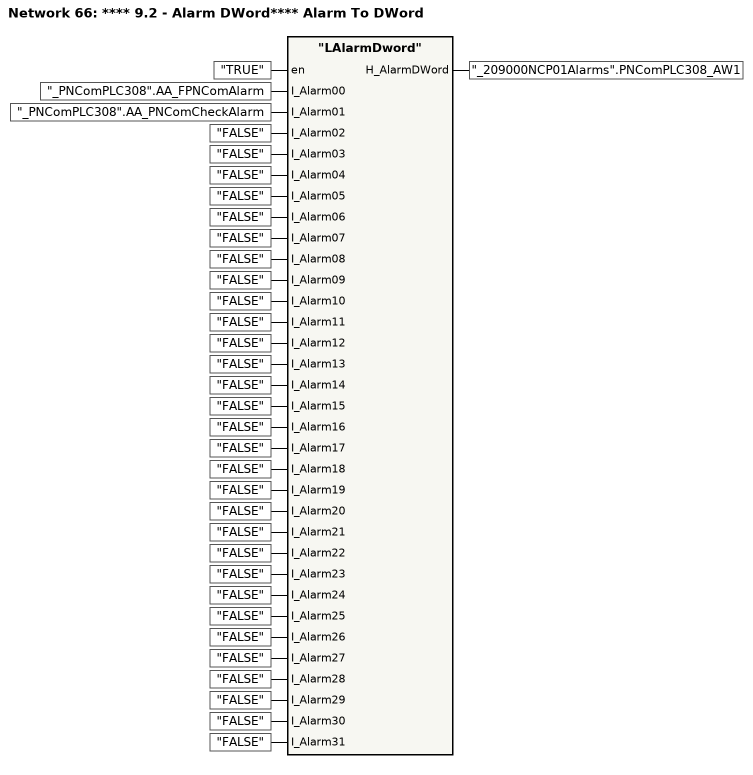
   IF "TRUE" THEN
       "LAlarmDword"(I_Alarm00 := "_PNComPLC308".AA_FPNComAlarm,
                     I_Alarm01 := "_PNComPLC308".AA_PNComCheckAlarm,
                     I_Alarm02 := "FALSE",
                     I_Alarm03 := "FALSE",
                     I_Alarm04 := "FALSE",
                     I_Alarm05 := "FALSE",
                     I_Alarm06 := "FALSE",
                     I_Alarm07 := "FALSE",
                     I_Alarm08 := "FALSE",
                     I_Alarm09 := "FALSE",
                     I_Alarm10 := "FALSE",
                     I_Alarm11 := "FALSE",
                     I_Alarm12 := "FALSE",
                     I_Alarm13 := "FALSE",
                     I_Alarm14 := "FALSE",
                     I_Alarm15 := "FALSE",
                     I_Alarm16 := "FALSE",
                     I_Alarm17 := "FALSE",
                     I_Alarm18 := "FALSE",
                     I_Alarm19 := "FALSE",
                     I_Alarm20 := "FALSE",
                     I_Alarm21 := "FALSE",
                     I_Alarm22 := "FALSE",
                     I_Alarm23 := "FALSE",
                     I_Alarm24 := "FALSE",
                     I_Alarm25 := "FALSE",
                     I_Alarm26 := "FALSE",
                     I_Alarm27 := "FALSE",
                     I_Alarm28 := "FALSE",
                     I_Alarm29 := "FALSE",
                     I_Alarm30 := "FALSE",
                     I_Alarm31 := "FALSE",
                     H_AlarmDWord => "_209000NCP01Alarms".PNComPLC308_AW1);
   END_IF;
END_REGION
END_FUNCTION
